TYPE ST_KPI_ItemsProduced :
STRUCT
	Total					: UDINT;
	Passed				: UDINT;
	Rejected				: UDINT;
	Efficiency				: LREAL;
	CreatedFiles			: UDINT;
	WarningLevel			: REAL := 99.75;
	AlarmLevel			: REAL := 99.50;
END_STRUCT
END_TYPE

(* stored: Version 1.1.0.1
   DUT ST_KPI_ItemsProduced: Id {71f64bb6-5fe6-4be1-8fc0-1b16dcf2b2bf} *)
